% RSLogix 500 project rev_pulse_monroe.RSS, saved by version 8.30.00.16 %
PROJECT "UNTITLED"    % processor: Bul.1763 MicroLogix 1100 Series B %

PROGRAM FILES
  LAD 2   4 rungs

DATA FILES
  O0 OUTPUT  4 elements
  I1 INPUT  6 elements
  S2 STATUS  66 elements
  B3 BINARY  24 elements
  T4 TIMER  1 elements
  C5 COUNTER  1 elements
  R6 CONTROL  1 elements
  N7 INTEGER  2 elements
  F8 FLOAT  10 elements
  L9 MISCELLANY  10 elements

LADDER 2
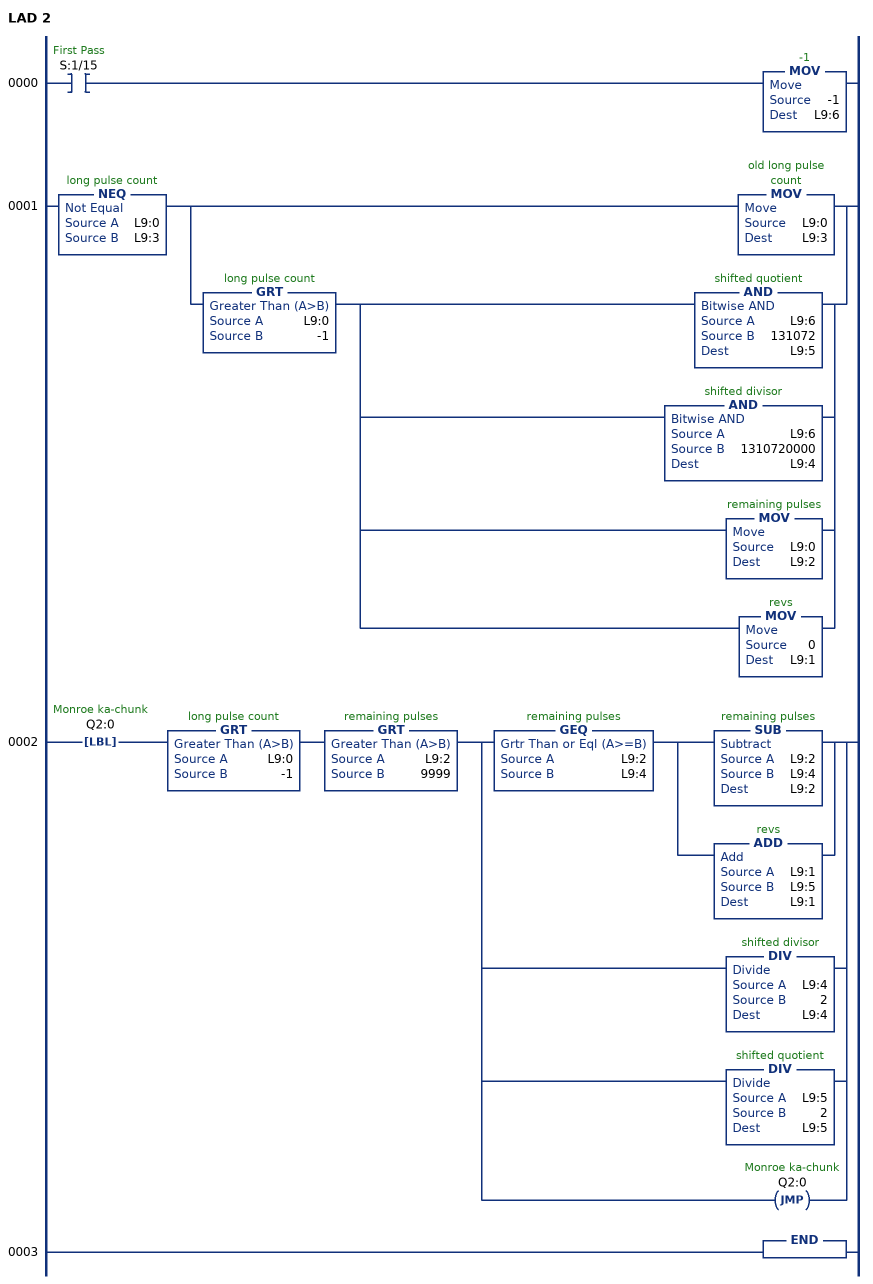
% Rung: 0 %
SOR XIC S:1/15 MOV -1 L9:6 EOR
%   S:1/15  "First Pass" %
%   L9:6  "-1" %
% Rung: 1 %
SOR NEQ L9:0 L9:3 BST MOV L9:0 L9:3 NXB GRT L9:0 -1 BST AND L9:6 131072 L9:5 NXB AND L9:6 1310720000 L9:4 NXB MOV L9:0 L9:2 NXB MOV 0 L9:1 BND BND EOR
%   L9:0  "long pulse count" %
%   L9:3  "old long pulse count" %
%   L9:6  "-1" %
%   L9:5  "shifted quotient" %
%   L9:4  "shifted divisor" %
%   L9:2  "remaining pulses" %
%   L9:1  "revs" %
% Rung: 2 %
SOR LBL Q2:0 GRT L9:0 -1 GRT L9:2 9999 BST GEQ L9:2 L9:4 BST SUB L9:2 L9:4 L9:2 NXB ADD L9:1 L9:5 L9:1 BND NXB DIV L9:4 2 L9:4 NXB DIV L9:5 2 L9:5 NXB JMP Q2:0 BND EOR
%   Q2:0  "Monroe ka-chunk" %
%   L9:0  "long pulse count" %
%   L9:2  "remaining pulses" %
%   L9:4  "shifted divisor" %
%   L9:1  "revs" %
%   L9:5  "shifted quotient" %
% Rung: 3 %
SOR END EOR

OTHER DOCUMENTED ADDRESSES
  B3:0/0  "disable math"
  F8:0  "float rev.pulse"
  S:22  S  "Maximum Observed Scan Time"
